// TIA Portal V17 export
// export: Created 2025-03-13T10:29:47.9061342Z, ExportSetting WithDefaults, DisplayName Totally Integrated Automation Portal, DisplayVersion V17 Update 8, DisplayName TIA Portal Openness, DisplayVersion V17 Update 8, DisplayName TIA Portal Version Control Interface, DisplayVersion V17, DisplayName SINAMICS Startdrive Advanced, DisplayVersion V17 SP2, DisplayName SINAMICS Startdrive G110M, G120, G120C, G120D, G120P, G115D, DisplayVersion V17 SP2, DisplayName SINAMICS Startdrive G130, G150, S120, S150, SINAMICS MV, S210, DisplayVersion V17 SP2, DisplayName STEP 7 Professional, DisplayVersion V17 Update 8, DisplayName SINUMERIK ONE STEP 7 Toolbox, DisplayVersion V17 Update 12, DisplayName SINUMERIK 840D sl STEP 7 Toolbox, DisplayVersion V17 Update 12, DisplayName STEP 7 Safety, DisplayVersion V17 Update 6, DisplayName WinCC Advanced, DisplayVersion V17 Update 8
FUNCTION "FC3610_U2_F2_GRIPPER" : Void   // FC3610, LAD
TITLE = FC2610_F2_GRIPPER
{ S7_Optimized_Access := 'FALSE' }
AUTHOR : ETXETAR
VERSION : 1.0
// stored: AutoNumber false, IsIECCheckEnabled false, SetENOAutomatically false, UDAEnableTagReadback false
   VAR_TEMP
      RET_VAL_1 : Int;
      UNIT_NUMBER : UInt;
      STATION_NUMBER : UInt;
   END_VAR
   VAR_TEMP   // added for the SCL form of the ladder/FBD networks
      _w1 : Bool;
   END_VAR
BEGIN

REGION Network 1: UNIT NUMBER AND STATION NUMBER DEFINITION
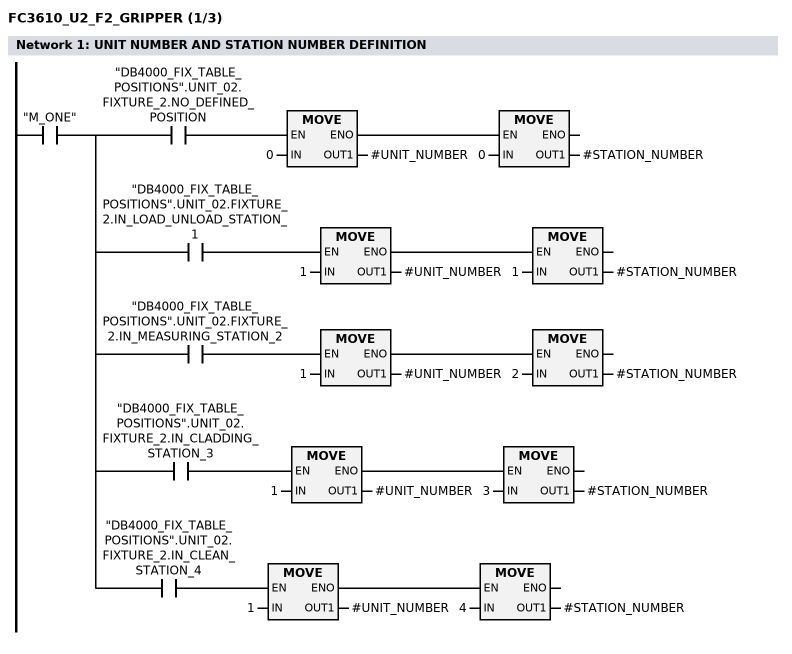
   RUNG wire#powerrail
      Contact( "M_ONE" )
      wire#w1
      Contact( "DB4000_FIX_TABLE_POSITIONS".UNIT_02.FIXTURE_2.NO_DEFINED_POSITION )
      Move(in := 0, out1 => #UNIT_NUMBER)
      Move(in := 0, out1 => #STATION_NUMBER)
   END_RUNG
   RUNG wire#w1
      Contact( "DB4000_FIX_TABLE_POSITIONS".UNIT_02.FIXTURE_2.IN_LOAD_UNLOAD_STATION_1 )
      Move(in := 1, out1 => #UNIT_NUMBER)
      Move(in := 1, out1 => #STATION_NUMBER)
   END_RUNG
   RUNG wire#w1
      Contact( "DB4000_FIX_TABLE_POSITIONS".UNIT_02.FIXTURE_2.IN_MEASURING_STATION_2 )
      Move(in := 1, out1 => #UNIT_NUMBER)
      Move(in := 2, out1 => #STATION_NUMBER)
   END_RUNG
   RUNG wire#w1
      Contact( "DB4000_FIX_TABLE_POSITIONS".UNIT_02.FIXTURE_2.IN_CLADDING_STATION_3 )
      Move(in := 1, out1 => #UNIT_NUMBER)
      Move(in := 3, out1 => #STATION_NUMBER)
   END_RUNG
   RUNG wire#w1
      Contact( "DB4000_FIX_TABLE_POSITIONS".UNIT_02.FIXTURE_2.IN_CLEAN_STATION_4 )
      Move(in := 1, out1 => #UNIT_NUMBER)
      Move(in := 4, out1 => #STATION_NUMBER)
   END_RUNG
   // the same network as SCL:
   IF "M_ONE" AND "DB4000_FIX_TABLE_POSITIONS".UNIT_02.FIXTURE_2.NO_DEFINED_POSITION THEN
       #UNIT_NUMBER := 0;
       #STATION_NUMBER := 0;
   END_IF;
   IF "M_ONE" AND "DB4000_FIX_TABLE_POSITIONS".UNIT_02.FIXTURE_2.IN_LOAD_UNLOAD_STATION_1 THEN
       #UNIT_NUMBER := 1;
       #STATION_NUMBER := 1;
   END_IF;
   IF "M_ONE" AND "DB4000_FIX_TABLE_POSITIONS".UNIT_02.FIXTURE_2.IN_MEASURING_STATION_2 THEN
       #UNIT_NUMBER := 1;
       #STATION_NUMBER := 2;
   END_IF;
   IF "M_ONE" AND "DB4000_FIX_TABLE_POSITIONS".UNIT_02.FIXTURE_2.IN_CLADDING_STATION_3 THEN
       #UNIT_NUMBER := 1;
       #STATION_NUMBER := 3;
   END_IF;
   IF "M_ONE" AND "DB4000_FIX_TABLE_POSITIONS".UNIT_02.FIXTURE_2.IN_CLEAN_STATION_4 THEN
       #UNIT_NUMBER := 1;
       #STATION_NUMBER := 4;
   END_IF;
END_REGION

REGION Network 2: CALL FB2509 FIXTURE 1 GRIPPER
   // 2#0000_0001 OPTIONS 0 BIT 0 LOCATED INPUT 1 OPTION
   // 2#0000_0010 OPTIONS 0 BIT 1 LOCATED INPUT 2 OPTION
   // 2#0000_0100 OPTIONS 0 BIT 2 LOCATED INPUT 3 OPTION
   // 2#0000_1000 OPTIONS 0 BIT 3 LOCATED INPUT 4 OPTION
   // 2#0001_0000 OPTIONS 0 BIT 4 LOCATED PRESSURE INPUT 1 OPTION
   // 2#0010_0000 OPTIONS 0 BIT 5 LOCATED PRESSURE INPUT 2 OPTION
   // 2#0100_0000 OPTIONS 0 BIT 6 LOW PRESSURE INPUT 1 OPTION
   // 2#1000_0000 OPTIONS 0 BIT 7 SPARE OPTION
   // 
   // 2#0000_0001 OPTIONS 1 BIT 0 RETURNED INPUT 1 OPTION
   // 2#0000_0010 OPTIONS 1 BIT 1 RETURNED INPUT 2 OPTION
   // 2#0000_0100 OPTIONS 1 BIT 2 RETURNED INPUT 3 OPTION
   // 2#0000_1000 OPTIONS 1 BIT 3 RETURNED INPUT 4 OPTION
   // 2#0001_0000 OPTIONS 1 BIT 4 RETURNED PRESSURE INPUT 1 OPTION
   // 2#0010_0000 OPTIONS 1 BIT 5 RETURNED PRESSURE INPUT 2 OPTION
   // 2#0100_0000 OPTIONS 1 BIT 6 SPARE OPTION
   // 2#1000_0000 OPTIONS 1 BIT 7 SPARE OPTION
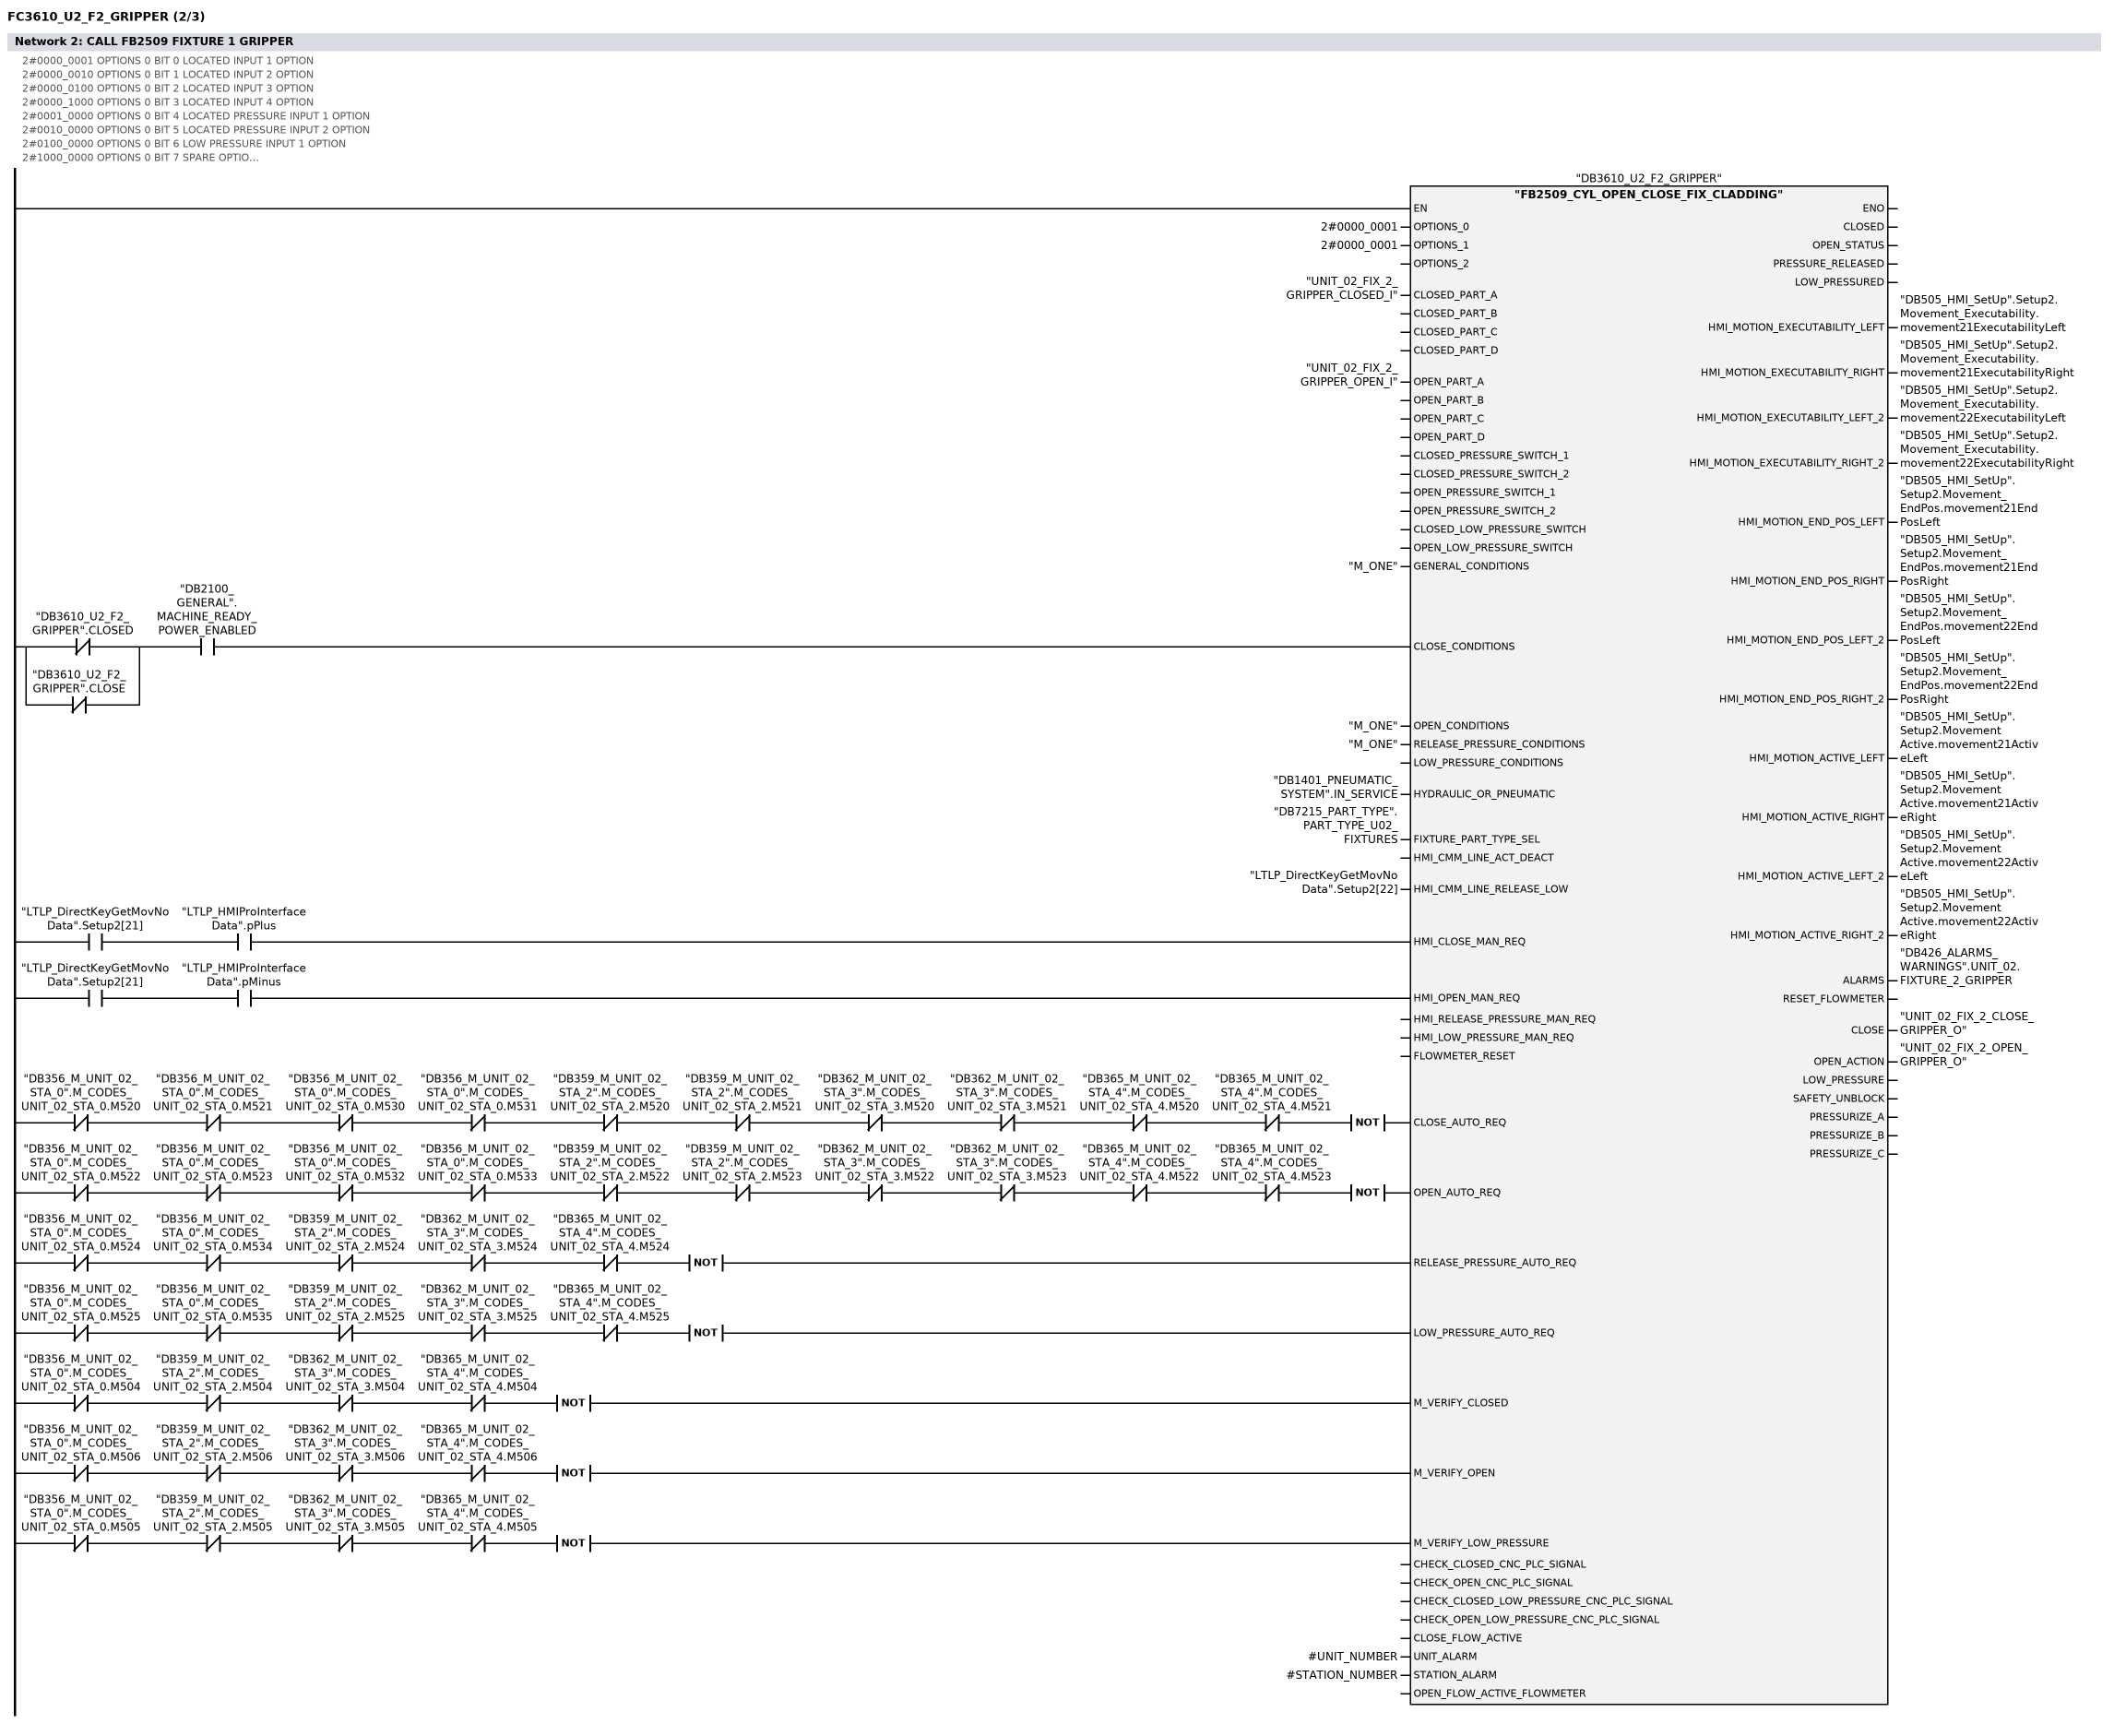
   RUNG wire#powerrail
      "DB3610_U2_F2_GRIPPER"(CLOSE_CONDITIONS := wire#w2, HMI_CLOSE_MAN_REQ := wire#w3, HMI_OPEN_MAN_REQ := wire#w4, CLOSE_AUTO_REQ := wire#w5, OPEN_AUTO_REQ := wire#w6, RELEASE_PRESSURE_AUTO_REQ := wire#w7, LOW_PRESSURE_AUTO_REQ := wire#w8, M_VERIFY_CLOSED := wire#w9, M_VERIFY_OPEN := wire#w10, M_VERIFY_LOW_PRESSURE := wire#w11, OPTIONS_0 := 2#0000_0001, OPTIONS_1 := 2#0000_0001, OPTIONS_2 :=, CLOSED_PART_A := "UNIT_02_FIX_2_GRIPPER_CLOSED_I", CLOSED_PART_B :=, CLOSED_PART_C :=, CLOSED_PART_D :=, OPEN_PART_A := "UNIT_02_FIX_2_GRIPPER_OPEN_I", OPEN_PART_B :=, OPEN_PART_C :=, OPEN_PART_D :=, CLOSED_PRESSURE_SWITCH_1 :=, CLOSED_PRESSURE_SWITCH_2 :=, OPEN_PRESSURE_SWITCH_1 :=, OPEN_PRESSURE_SWITCH_2 :=, CLOSED_LOW_PRESSURE_SWITCH :=, OPEN_LOW_PRESSURE_SWITCH :=, GENERAL_CONDITIONS := "M_ONE", OPEN_CONDITIONS := "M_ONE", RELEASE_PRESSURE_CONDITIONS := "M_ONE", LOW_PRESSURE_CONDITIONS :=, HYDRAULIC_OR_PNEUMATIC := "DB1401_PNEUMATIC_SYSTEM".IN_SERVICE, FIXTURE_PART_TYPE_SEL := "DB7215_PART_TYPE".PART_TYPE_U02_FIXTURES, HMI_CMM_LINE_ACT_DEACT :=, HMI_CMM_LINE_RELEASE_LOW := "LTLP_DirectKeyGetMovNoData".Setup2[22], HMI_RELEASE_PRESSURE_MAN_REQ :=, HMI_LOW_PRESSURE_MAN_REQ :=, FLOWMETER_RESET :=, CHECK_CLOSED_CNC_PLC_SIGNAL :=, CHECK_OPEN_CNC_PLC_SIGNAL :=, CHECK_CLOSED_LOW_PRESSURE_CNC_PLC_SIGNAL :=, CHECK_OPEN_LOW_PRESSURE_CNC_PLC_SIGNAL :=, CLOSE_FLOW_ACTIVE :=, UNIT_ALARM := #UNIT_NUMBER, STATION_ALARM := #STATION_NUMBER, OPEN_FLOW_ACTIVE_FLOWMETER :=, CLOSED =>, OPEN_STATUS =>, PRESSURE_RELEASED =>, LOW_PRESSURED =>, HMI_MOTION_EXECUTABILITY_LEFT => "DB505_HMI_SetUp".Setup2.Movement_Executability.movement21ExecutabilityLeft, HMI_MOTION_EXECUTABILITY_RIGHT => "DB505_HMI_SetUp".Setup2.Movement_Executability.movement21ExecutabilityRight, HMI_MOTION_EXECUTABILITY_LEFT_2 => "DB505_HMI_SetUp".Setup2.Movement_Executability.movement22ExecutabilityLeft, HMI_MOTION_EXECUTABILITY_RIGHT_2 => "DB505_HMI_SetUp".Setup2.Movement_Executability.movement22ExecutabilityRight, HMI_MOTION_END_POS_LEFT => "DB505_HMI_SetUp".Setup2.Movement_EndPos.movement21EndPosLeft, HMI_MOTION_END_POS_RIGHT => "DB505_HMI_SetUp".Setup2.Movement_EndPos.movement21EndPosRight, HMI_MOTION_END_POS_LEFT_2 => "DB505_HMI_SetUp".Setup2.Movement_EndPos.movement22EndPosLeft, HMI_MOTION_END_POS_RIGHT_2 => "DB505_HMI_SetUp".Setup2.Movement_EndPos.movement22EndPosRight, HMI_MOTION_ACTIVE_LEFT => "DB505_HMI_SetUp".Setup2.MovementActive.movement21ActiveLeft, HMI_MOTION_ACTIVE_RIGHT => "DB505_HMI_SetUp".Setup2.MovementActive.movement21ActiveRight, HMI_MOTION_ACTIVE_LEFT_2 => "DB505_HMI_SetUp".Setup2.MovementActive.movement22ActiveLeft, HMI_MOTION_ACTIVE_RIGHT_2 => "DB505_HMI_SetUp".Setup2.MovementActive.movement22ActiveRight, ALARMS => "DB426_ALARMS_WARNINGS".UNIT_02.FIXTURE_2_GRIPPER, RESET_FLOWMETER =>, CLOSE => "UNIT_02_FIX_2_CLOSE_GRIPPER_O", OPEN_ACTION => "UNIT_02_FIX_2_OPEN_GRIPPER_O", LOW_PRESSURE =>, SAFETY_UNBLOCK =>, PRESSURIZE_A =>, PRESSURIZE_B =>, PRESSURIZE_C =>)
   END_RUNG
   RUNG wire#powerrail
      I_Contact( "DB3610_U2_F2_GRIPPER".CLOSED )
      wire#w1
      Contact( "DB2100_GENERAL".MACHINE_READY_POWER_ENABLED )
   END_RUNG wire#w2
   RUNG wire#powerrail
      I_Contact( "DB3610_U2_F2_GRIPPER".CLOSE )
   END_RUNG wire#w1
   RUNG wire#powerrail
      Contact( "LTLP_DirectKeyGetMovNoData".Setup2[21] )
      Contact( "LTLP_HMIProInterfaceData".pPlus )
   END_RUNG wire#w3
   RUNG wire#powerrail
      Contact( "LTLP_DirectKeyGetMovNoData".Setup2[21] )
      Contact( "LTLP_HMIProInterfaceData".pMinus )
   END_RUNG wire#w4
   RUNG wire#powerrail
      I_Contact( "DB356_M_UNIT_02_STA_0".M_CODES_UNIT_02_STA_0.M520 )
      I_Contact( "DB356_M_UNIT_02_STA_0".M_CODES_UNIT_02_STA_0.M521 )
      I_Contact( "DB356_M_UNIT_02_STA_0".M_CODES_UNIT_02_STA_0.M530 )
      I_Contact( "DB356_M_UNIT_02_STA_0".M_CODES_UNIT_02_STA_0.M531 )
      I_Contact( "DB359_M_UNIT_02_STA_2".M_CODES_UNIT_02_STA_2.M520 )
      I_Contact( "DB359_M_UNIT_02_STA_2".M_CODES_UNIT_02_STA_2.M521 )
      I_Contact( "DB362_M_UNIT_02_STA_3".M_CODES_UNIT_02_STA_3.M520 )
      I_Contact( "DB362_M_UNIT_02_STA_3".M_CODES_UNIT_02_STA_3.M521 )
      I_Contact( "DB365_M_UNIT_02_STA_4".M_CODES_UNIT_02_STA_4.M520 )
      I_Contact( "DB365_M_UNIT_02_STA_4".M_CODES_UNIT_02_STA_4.M521 )
      Not()
   END_RUNG wire#w5
   RUNG wire#powerrail
      I_Contact( "DB356_M_UNIT_02_STA_0".M_CODES_UNIT_02_STA_0.M522 )
      I_Contact( "DB356_M_UNIT_02_STA_0".M_CODES_UNIT_02_STA_0.M523 )
      I_Contact( "DB356_M_UNIT_02_STA_0".M_CODES_UNIT_02_STA_0.M532 )
      I_Contact( "DB356_M_UNIT_02_STA_0".M_CODES_UNIT_02_STA_0.M533 )
      I_Contact( "DB359_M_UNIT_02_STA_2".M_CODES_UNIT_02_STA_2.M522 )
      I_Contact( "DB359_M_UNIT_02_STA_2".M_CODES_UNIT_02_STA_2.M523 )
      I_Contact( "DB362_M_UNIT_02_STA_3".M_CODES_UNIT_02_STA_3.M522 )
      I_Contact( "DB362_M_UNIT_02_STA_3".M_CODES_UNIT_02_STA_3.M523 )
      I_Contact( "DB365_M_UNIT_02_STA_4".M_CODES_UNIT_02_STA_4.M522 )
      I_Contact( "DB365_M_UNIT_02_STA_4".M_CODES_UNIT_02_STA_4.M523 )
      Not()
   END_RUNG wire#w6
   RUNG wire#powerrail
      I_Contact( "DB356_M_UNIT_02_STA_0".M_CODES_UNIT_02_STA_0.M524 )
      I_Contact( "DB356_M_UNIT_02_STA_0".M_CODES_UNIT_02_STA_0.M534 )
      I_Contact( "DB359_M_UNIT_02_STA_2".M_CODES_UNIT_02_STA_2.M524 )
      I_Contact( "DB362_M_UNIT_02_STA_3".M_CODES_UNIT_02_STA_3.M524 )
      I_Contact( "DB365_M_UNIT_02_STA_4".M_CODES_UNIT_02_STA_4.M524 )
      Not()
   END_RUNG wire#w7
   RUNG wire#powerrail
      I_Contact( "DB356_M_UNIT_02_STA_0".M_CODES_UNIT_02_STA_0.M525 )
      I_Contact( "DB356_M_UNIT_02_STA_0".M_CODES_UNIT_02_STA_0.M535 )
      I_Contact( "DB359_M_UNIT_02_STA_2".M_CODES_UNIT_02_STA_2.M525 )
      I_Contact( "DB362_M_UNIT_02_STA_3".M_CODES_UNIT_02_STA_3.M525 )
      I_Contact( "DB365_M_UNIT_02_STA_4".M_CODES_UNIT_02_STA_4.M525 )
      Not()
   END_RUNG wire#w8
   RUNG wire#powerrail
      I_Contact( "DB356_M_UNIT_02_STA_0".M_CODES_UNIT_02_STA_0.M504 )
      I_Contact( "DB359_M_UNIT_02_STA_2".M_CODES_UNIT_02_STA_2.M504 )
      I_Contact( "DB362_M_UNIT_02_STA_3".M_CODES_UNIT_02_STA_3.M504 )
      I_Contact( "DB365_M_UNIT_02_STA_4".M_CODES_UNIT_02_STA_4.M504 )
      Not()
   END_RUNG wire#w9
   RUNG wire#powerrail
      I_Contact( "DB356_M_UNIT_02_STA_0".M_CODES_UNIT_02_STA_0.M506 )
      I_Contact( "DB359_M_UNIT_02_STA_2".M_CODES_UNIT_02_STA_2.M506 )
      I_Contact( "DB362_M_UNIT_02_STA_3".M_CODES_UNIT_02_STA_3.M506 )
      I_Contact( "DB365_M_UNIT_02_STA_4".M_CODES_UNIT_02_STA_4.M506 )
      Not()
   END_RUNG wire#w10
   RUNG wire#powerrail
      I_Contact( "DB356_M_UNIT_02_STA_0".M_CODES_UNIT_02_STA_0.M505 )
      I_Contact( "DB359_M_UNIT_02_STA_2".M_CODES_UNIT_02_STA_2.M505 )
      I_Contact( "DB362_M_UNIT_02_STA_3".M_CODES_UNIT_02_STA_3.M505 )
      I_Contact( "DB365_M_UNIT_02_STA_4".M_CODES_UNIT_02_STA_4.M505 )
      Not()
   END_RUNG wire#w11
   // the same network as SCL:
   "DB3610_U2_F2_GRIPPER"(OPTIONS_0 := 2#0000_0001,   // "FB2509_CYL_OPEN_CLOSE_FIX_CLADDING"
                          OPTIONS_1 := 2#0000_0001,
                          CLOSED_PART_A := "UNIT_02_FIX_2_GRIPPER_CLOSED_I",
                          OPEN_PART_A := "UNIT_02_FIX_2_GRIPPER_OPEN_I",
                          GENERAL_CONDITIONS := "M_ONE",
                          CLOSE_CONDITIONS := (NOT "DB3610_U2_F2_GRIPPER".CLOSED OR NOT "DB3610_U2_F2_GRIPPER".CLOSE) AND "DB2100_GENERAL".MACHINE_READY_POWER_ENABLED,
                          OPEN_CONDITIONS := "M_ONE",
                          RELEASE_PRESSURE_CONDITIONS := "M_ONE",
                          HYDRAULIC_OR_PNEUMATIC := "DB1401_PNEUMATIC_SYSTEM".IN_SERVICE,
                          FIXTURE_PART_TYPE_SEL := "DB7215_PART_TYPE".PART_TYPE_U02_FIXTURES,
                          HMI_CMM_LINE_RELEASE_LOW := "LTLP_DirectKeyGetMovNoData".Setup2[22],
                          HMI_CLOSE_MAN_REQ := "LTLP_DirectKeyGetMovNoData".Setup2[21] AND "LTLP_HMIProInterfaceData".pPlus,
                          HMI_OPEN_MAN_REQ := "LTLP_DirectKeyGetMovNoData".Setup2[21] AND "LTLP_HMIProInterfaceData".pMinus,
                          CLOSE_AUTO_REQ := NOT (NOT "DB356_M_UNIT_02_STA_0".M_CODES_UNIT_02_STA_0.M520 AND NOT "DB356_M_UNIT_02_STA_0".M_CODES_UNIT_02_STA_0.M521 AND NOT "DB356_M_UNIT_02_STA_0".M_CODES_UNIT_02_STA_0.M530 AND NOT "DB356_M_UNIT_02_STA_0".M_CODES_UNIT_02_STA_0.M531 AND NOT "DB359_M_UNIT_02_STA_2".M_CODES_UNIT_02_STA_2.M520 AND NOT "DB359_M_UNIT_02_STA_2".M_CODES_UNIT_02_STA_2.M521 AND NOT "DB362_M_UNIT_02_STA_3".M_CODES_UNIT_02_STA_3.M520 AND NOT "DB362_M_UNIT_02_STA_3".M_CODES_UNIT_02_STA_3.M521 AND NOT "DB365_M_UNIT_02_STA_4".M_CODES_UNIT_02_STA_4.M520 AND NOT "DB365_M_UNIT_02_STA_4".M_CODES_UNIT_02_STA_4.M521),
                          OPEN_AUTO_REQ := NOT (NOT "DB356_M_UNIT_02_STA_0".M_CODES_UNIT_02_STA_0.M522 AND NOT "DB356_M_UNIT_02_STA_0".M_CODES_UNIT_02_STA_0.M523 AND NOT "DB356_M_UNIT_02_STA_0".M_CODES_UNIT_02_STA_0.M532 AND NOT "DB356_M_UNIT_02_STA_0".M_CODES_UNIT_02_STA_0.M533 AND NOT "DB359_M_UNIT_02_STA_2".M_CODES_UNIT_02_STA_2.M522 AND NOT "DB359_M_UNIT_02_STA_2".M_CODES_UNIT_02_STA_2.M523 AND NOT "DB362_M_UNIT_02_STA_3".M_CODES_UNIT_02_STA_3.M522 AND NOT "DB362_M_UNIT_02_STA_3".M_CODES_UNIT_02_STA_3.M523 AND NOT "DB365_M_UNIT_02_STA_4".M_CODES_UNIT_02_STA_4.M522 AND NOT "DB365_M_UNIT_02_STA_4".M_CODES_UNIT_02_STA_4.M523),
                          RELEASE_PRESSURE_AUTO_REQ := NOT (NOT "DB356_M_UNIT_02_STA_0".M_CODES_UNIT_02_STA_0.M524 AND NOT "DB356_M_UNIT_02_STA_0".M_CODES_UNIT_02_STA_0.M534 AND NOT "DB359_M_UNIT_02_STA_2".M_CODES_UNIT_02_STA_2.M524 AND NOT "DB362_M_UNIT_02_STA_3".M_CODES_UNIT_02_STA_3.M524 AND NOT "DB365_M_UNIT_02_STA_4".M_CODES_UNIT_02_STA_4.M524),
                          LOW_PRESSURE_AUTO_REQ := NOT (NOT "DB356_M_UNIT_02_STA_0".M_CODES_UNIT_02_STA_0.M525 AND NOT "DB356_M_UNIT_02_STA_0".M_CODES_UNIT_02_STA_0.M535 AND NOT "DB359_M_UNIT_02_STA_2".M_CODES_UNIT_02_STA_2.M525 AND NOT "DB362_M_UNIT_02_STA_3".M_CODES_UNIT_02_STA_3.M525 AND NOT "DB365_M_UNIT_02_STA_4".M_CODES_UNIT_02_STA_4.M525),
                          M_VERIFY_CLOSED := NOT (NOT "DB356_M_UNIT_02_STA_0".M_CODES_UNIT_02_STA_0.M504 AND NOT "DB359_M_UNIT_02_STA_2".M_CODES_UNIT_02_STA_2.M504 AND NOT "DB362_M_UNIT_02_STA_3".M_CODES_UNIT_02_STA_3.M504 AND NOT "DB365_M_UNIT_02_STA_4".M_CODES_UNIT_02_STA_4.M504),
                          M_VERIFY_OPEN := NOT (NOT "DB356_M_UNIT_02_STA_0".M_CODES_UNIT_02_STA_0.M506 AND NOT "DB359_M_UNIT_02_STA_2".M_CODES_UNIT_02_STA_2.M506 AND NOT "DB362_M_UNIT_02_STA_3".M_CODES_UNIT_02_STA_3.M506 AND NOT "DB365_M_UNIT_02_STA_4".M_CODES_UNIT_02_STA_4.M506),
                          M_VERIFY_LOW_PRESSURE := NOT (NOT "DB356_M_UNIT_02_STA_0".M_CODES_UNIT_02_STA_0.M505 AND NOT "DB359_M_UNIT_02_STA_2".M_CODES_UNIT_02_STA_2.M505 AND NOT "DB362_M_UNIT_02_STA_3".M_CODES_UNIT_02_STA_3.M505 AND NOT "DB365_M_UNIT_02_STA_4".M_CODES_UNIT_02_STA_4.M505),
                          UNIT_ALARM := #UNIT_NUMBER,
                          STATION_ALARM := #STATION_NUMBER,
                          HMI_MOTION_EXECUTABILITY_LEFT => "DB505_HMI_SetUp".Setup2.Movement_Executability.movement21ExecutabilityLeft,
                          HMI_MOTION_EXECUTABILITY_RIGHT => "DB505_HMI_SetUp".Setup2.Movement_Executability.movement21ExecutabilityRight,
                          HMI_MOTION_EXECUTABILITY_LEFT_2 => "DB505_HMI_SetUp".Setup2.Movement_Executability.movement22ExecutabilityLeft,
                          HMI_MOTION_EXECUTABILITY_RIGHT_2 => "DB505_HMI_SetUp".Setup2.Movement_Executability.movement22ExecutabilityRight,
                          HMI_MOTION_END_POS_LEFT => "DB505_HMI_SetUp".Setup2.Movement_EndPos.movement21EndPosLeft,
                          HMI_MOTION_END_POS_RIGHT => "DB505_HMI_SetUp".Setup2.Movement_EndPos.movement21EndPosRight,
                          HMI_MOTION_END_POS_LEFT_2 => "DB505_HMI_SetUp".Setup2.Movement_EndPos.movement22EndPosLeft,
                          HMI_MOTION_END_POS_RIGHT_2 => "DB505_HMI_SetUp".Setup2.Movement_EndPos.movement22EndPosRight,
                          HMI_MOTION_ACTIVE_LEFT => "DB505_HMI_SetUp".Setup2.MovementActive.movement21ActiveLeft,
                          HMI_MOTION_ACTIVE_RIGHT => "DB505_HMI_SetUp".Setup2.MovementActive.movement21ActiveRight,
                          HMI_MOTION_ACTIVE_LEFT_2 => "DB505_HMI_SetUp".Setup2.MovementActive.movement22ActiveLeft,
                          HMI_MOTION_ACTIVE_RIGHT_2 => "DB505_HMI_SetUp".Setup2.MovementActive.movement22ActiveRight,
                          ALARMS => "DB426_ALARMS_WARNINGS".UNIT_02.FIXTURE_2_GRIPPER,
                          CLOSE => "UNIT_02_FIX_2_CLOSE_GRIPPER_O",
                          OPEN_ACTION => "UNIT_02_FIX_2_OPEN_GRIPPER_O");
END_REGION

REGION Network 3: OPERATOR HELP
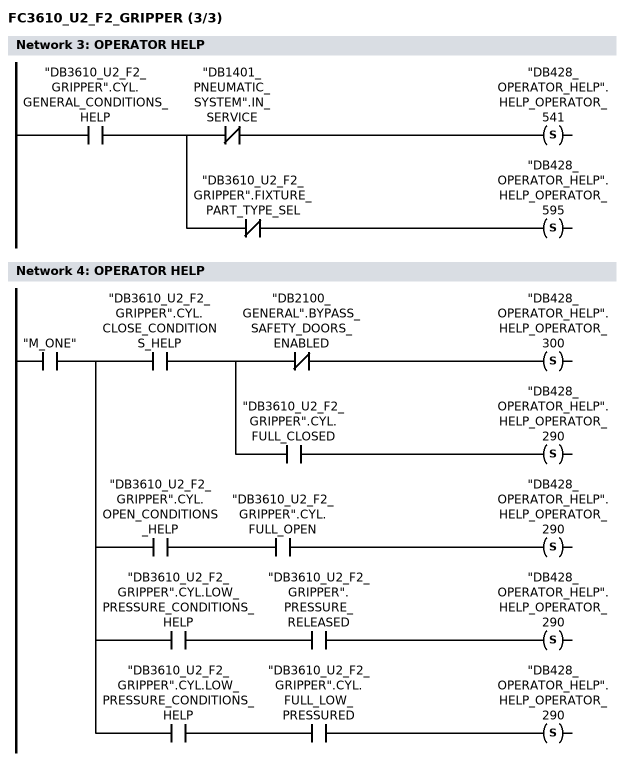
   RUNG wire#powerrail
      Contact( "DB3610_U2_F2_GRIPPER".CYL.GENERAL_CONDITIONS_HELP )
      wire#w1
      I_Contact( "DB1401_PNEUMATIC_SYSTEM".IN_SERVICE )
      S_Coil( "DB428_OPERATOR_HELP".HELP_OPERATOR_541 )
   END_RUNG
   RUNG wire#w1
      I_Contact( "DB3610_U2_F2_GRIPPER".FIXTURE_PART_TYPE_SEL )
      S_Coil( "DB428_OPERATOR_HELP".HELP_OPERATOR_595 )
   END_RUNG
   // the same network as SCL:
   IF "DB3610_U2_F2_GRIPPER".CYL.GENERAL_CONDITIONS_HELP AND NOT "DB1401_PNEUMATIC_SYSTEM".IN_SERVICE THEN
       "DB428_OPERATOR_HELP".HELP_OPERATOR_541 := TRUE;
   END_IF;
   IF "DB3610_U2_F2_GRIPPER".CYL.GENERAL_CONDITIONS_HELP AND NOT "DB3610_U2_F2_GRIPPER".FIXTURE_PART_TYPE_SEL THEN
       "DB428_OPERATOR_HELP".HELP_OPERATOR_595 := TRUE;
   END_IF;
END_REGION

REGION Network 4: OPERATOR HELP
   RUNG wire#powerrail
      Contact( "M_ONE" )
      wire#w1
      Contact( "DB3610_U2_F2_GRIPPER".CYL.CLOSE_CONDITIONS_HELP )
      wire#w2
      I_Contact( "DB2100_GENERAL".BYPASS_SAFETY_DOORS_ENABLED )
      S_Coil( "DB428_OPERATOR_HELP".HELP_OPERATOR_300 )
   END_RUNG
   RUNG wire#w2
      Contact( "DB3610_U2_F2_GRIPPER".CYL.FULL_CLOSED )
      S_Coil( "DB428_OPERATOR_HELP".HELP_OPERATOR_290 )
   END_RUNG
   RUNG wire#w1
      Contact( "DB3610_U2_F2_GRIPPER".CYL.OPEN_CONDITIONS_HELP )
      Contact( "DB3610_U2_F2_GRIPPER".CYL.FULL_OPEN )
      S_Coil( "DB428_OPERATOR_HELP".HELP_OPERATOR_290 )
   END_RUNG
   RUNG wire#w1
      Contact( "DB3610_U2_F2_GRIPPER".CYL.LOW_PRESSURE_CONDITIONS_HELP )
      Contact( "DB3610_U2_F2_GRIPPER".PRESSURE_RELEASED )
      S_Coil( "DB428_OPERATOR_HELP".HELP_OPERATOR_290 )
   END_RUNG
   RUNG wire#w1
      Contact( "DB3610_U2_F2_GRIPPER".CYL.LOW_PRESSURE_CONDITIONS_HELP )
      Contact( "DB3610_U2_F2_GRIPPER".CYL.FULL_LOW_PRESSURED )
      S_Coil( "DB428_OPERATOR_HELP".HELP_OPERATOR_290 )
   END_RUNG
   // the same network as SCL:
   #_w1 := "M_ONE" AND "DB3610_U2_F2_GRIPPER".CYL.CLOSE_CONDITIONS_HELP;
   IF #_w1 AND NOT "DB2100_GENERAL".BYPASS_SAFETY_DOORS_ENABLED THEN
       "DB428_OPERATOR_HELP".HELP_OPERATOR_300 := TRUE;
   END_IF;
   IF #_w1 AND "DB3610_U2_F2_GRIPPER".CYL.FULL_CLOSED THEN
       "DB428_OPERATOR_HELP".HELP_OPERATOR_290 := TRUE;
   END_IF;
   IF "M_ONE" AND "DB3610_U2_F2_GRIPPER".CYL.OPEN_CONDITIONS_HELP AND "DB3610_U2_F2_GRIPPER".CYL.FULL_OPEN THEN
       "DB428_OPERATOR_HELP".HELP_OPERATOR_290 := TRUE;
   END_IF;
   IF "M_ONE" AND "DB3610_U2_F2_GRIPPER".CYL.LOW_PRESSURE_CONDITIONS_HELP AND "DB3610_U2_F2_GRIPPER".PRESSURE_RELEASED THEN
       "DB428_OPERATOR_HELP".HELP_OPERATOR_290 := TRUE;
   END_IF;
   IF "M_ONE" AND "DB3610_U2_F2_GRIPPER".CYL.LOW_PRESSURE_CONDITIONS_HELP AND "DB3610_U2_F2_GRIPPER".CYL.FULL_LOW_PRESSURED THEN
       "DB428_OPERATOR_HELP".HELP_OPERATOR_290 := TRUE;
   END_IF;
END_REGION
END_FUNCTION
